// Mitsubishi GX Works2 project: 02fb   PLC: Q03UDV

// task Task_01 (event TRUE, interval 0, priority 31): POU_01
// task st_teste (event TRUE, interval 0, priority 31): st_teste

PROGRAM POU_01
VAR
  CTD_2 : CTD;
  CTU_1 : CTU;
  CTU_2 : CTU;
  R_TRIG_2 : R_TRIG;
  TP_1 : TP;
  TOF_1 : TOF;
  TON_1 : TON;
  timeon : TIME;
  timeof : TIME;
  timetp : TIME;
  TOF_2 : TOF;
  timeof2 : TIME;
  TON_2 : TON;
  timeon2 : TIME;
  TOF_3 : TOF;
  timeof3 : TIME;
  TP_2 : TP;
  TP_3 : TP;
  timept2 : TIME;
  timetp3 : TIME;
  bitOn : BOOL;
  bitOf : BOOL;
  TON_3 : TON;
  TON_4 : TON;
  TON_8 : TON;
  TON5 : TON;
  TOn10 : TON;
  TON_5 : TON;
  timeon5 : TIME;
  timeon3 : TIME;
  TON_6 : TON;
  timeon6 : TIME;
  TOF_4 : TOF;
  timeof7 : TIME;
  verde : BOOL;
  amarelo : BOOL;
  vermelho : BOOL;
  fbBlinker_1 : fbBlinker;
  fbBlinker_2 : fbBlinker;
  diResult : DINT;
  fbBlinker_3 : fbBlinker;
  result : INT;
  funOperacoes_1 : funOperacoes;
  resultS : ARRAY [0..1] OF INT;
  rseultSu : ARRAY [0..1] OF INT;
  resultM : ARRAY [0..1] OF INT;
  resultD : INT;
  resultSo : INT;
  rseultSub : ARRAY [0..1] OF INT;
  resultMult : ARRAY [0..1] OF INT;
  resultMulti : ARRAY [0..1] OF INT;
  resultMultiplicacao : ARRAY [0..1] OF INT;
  resultMUT : ARRAY [0..1] OF INT;
  rseultaSub : ARRAY [0..1] OF INT;
  resultadoSub : ARRAY [0..1] OF INT;
  resultadoMULt : ARRAY [0..1] OF INT;
  Subres : ARRAY [0..1] OF INT;
  Sres : INT;
  Splica : DINT;
  DIVIVALOR : INT;
  Dre : ARRAY [0..1] OF INT;
  habilitar : BOOL;
  valor1 : INT;
  valor2 : INT;
  tipOper : STRING[32];
END_VAR
(* structured ladder/FBD written out as ST: instructions are called as NAME(EN, inputs, outputs); _pN, _eN, _tN stand for wires *)
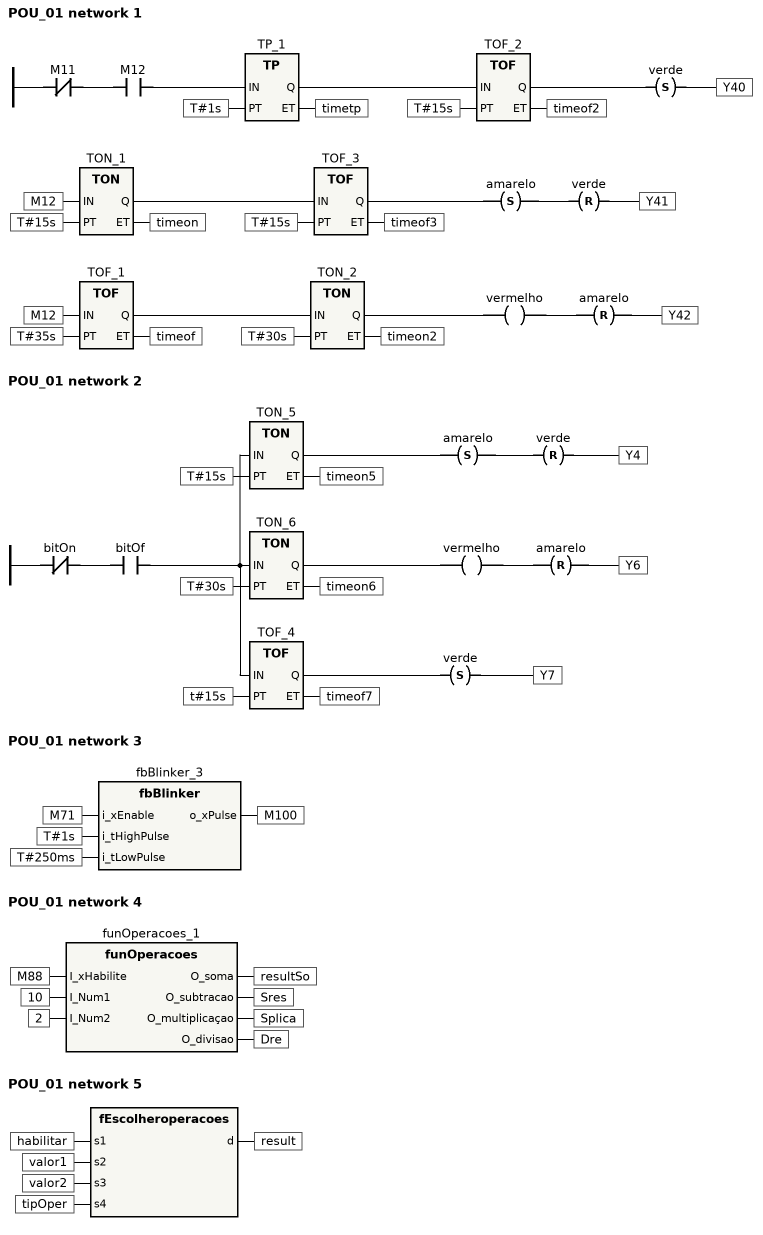
(* network 1 *)
TP_1(IN := NOT M11 AND M12, PT := T#1s, ET => timetp);
TOF_2(IN := TP_1.Q, PT := T#15s, ET => timeof2);
SET(TOF_2.Q, verde);
Y40 := TOF_2.Q;
TON_1(IN := M12, PT := T#15s, ET => timeon);
TOF_3(IN := TON_1.Q, PT := T#15s, ET => timeof3);
SET(TOF_3.Q, amarelo);
RST(TOF_3.Q, verde);
Y41 := TOF_3.Q;
TOF_1(IN := M12, PT := T#35s, ET => timeof);
TON_2(IN := TOF_1.Q, PT := T#30s, ET => timeon2);
vermelho := TON_2.Q;
RST(TON_2.Q, amarelo);
Y42 := TON_2.Q;
(* network 2 *)
_p1 := NOT bitOn AND bitOf;
TOF_4(IN := _p1, PT := t#15s, ET => timeof7);
SET(TOF_4.Q, verde);
Y7 := TOF_4.Q;
TON_5(IN := _p1, PT := T#15s, ET => timeon5);
SET(TON_5.Q, amarelo);
RST(TON_5.Q, verde);
Y4 := TON_5.Q;
TON_6(IN := _p1, PT := T#30s, ET => timeon6);
vermelho := TON_6.Q;
RST(TON_6.Q, amarelo);
Y6 := TON_6.Q;
(* network 3 *)
fbBlinker_3(i_xEnable := M71, i_tHighPulse := T#1s, i_tLowPulse := T#250ms, o_xPulse => M100);
(* network 4 *)
funOperacoes_1(I_xHabilite := M88, I_Num1 := 10, I_Num2 := 2, O_soma => resultSo, O_subtracao => Sres, O_multiplicaçao => Splica, O_divisao => Dre);
(* network 5 *)
result := fEscolheroperacoes(habilitar, valor1, valor2, tipOper);
END_PROGRAM

FUNCTION fSomaInt
VAR_INPUT
  I_xHabilitar : BOOL;
  I_Elemento1 : INT;
  I_Elemento2 : INT;
END_VAR
(* structured ladder/FBD written out as ST: instructions are called as NAME(EN, inputs, outputs); _pN, _eN, _tN stand for wires *)
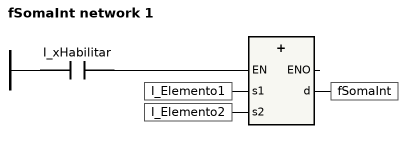
(* network 1 *)
+(I_xHabilitar, I_Elemento1, I_Elemento2, fSomaInt);
END_FUNCTION

FUNCTION fSubtracaoInt
VAR_INPUT
  I_xHabilitarS : BOOL;
  I_Elemento1S : INT;
  I_Elemento2S : INT;
END_VAR
(* structured ladder/FBD written out as ST: instructions are called as NAME(EN, inputs, outputs); _pN, _eN, _tN stand for wires *)
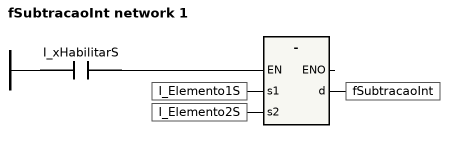
(* network 1 *)
-(I_xHabilitarS, I_Elemento1S, I_Elemento2S, fSubtracaoInt);
END_FUNCTION

FUNCTION_BLOCK fbBlinker
VAR_INPUT
  i_xEnable : BOOL;
  i_tHighPulse : TIME;
  i_tLowPulse : TIME;
END_VAR
VAR_OUTPUT
  o_xPulse : BOOL;
END_VAR
VAR
  fb_TimerHigh : TP;
  fb_TimerLow : TOF;
  xAuxiliar : BOOL;
END_VAR
(* structured ladder/FBD written out as ST: instructions are called as NAME(EN, inputs, outputs); _pN, _eN, _tN stand for wires *)
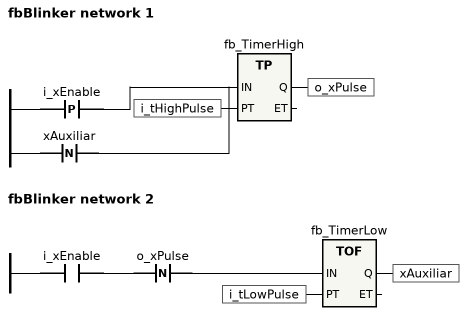
(* network 1 *)
fb_TimerHigh(IN := LDP(TRUE, i_xEnable) OR LDF(TRUE, xAuxiliar), PT := i_tHighPulse, Q => o_xPulse);
(* network 2 *)
fb_TimerLow(IN := i_xEnable AND LDF(TRUE, o_xPulse), PT := i_tLowPulse, Q => xAuxiliar);
END_FUNCTION_BLOCK

FUNCTION fMultInt
VAR_INPUT
  I_xHabilitar : BOOL;
  I_Elemento1 : INT;
  I_Elemento2 : INT;
END_VAR
(* structured ladder/FBD written out as ST: instructions are called as NAME(EN, inputs, outputs); _pN, _eN, _tN stand for wires *)
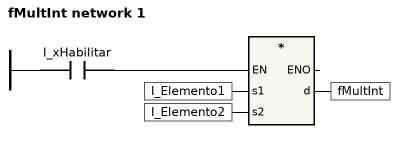
(* network 1 *)
*(I_xHabilitar, I_Elemento1, I_Elemento2, fMultInt);
END_FUNCTION

FUNCTION fDivisaoInt
VAR_INPUT
  I_xHabilitar : BOOL;
  I_Elemento1 : INT;
  I_Elemento2 : INT;
END_VAR
(* structured ladder/FBD written out as ST: instructions are called as NAME(EN, inputs, outputs); _pN, _eN, _tN stand for wires *)
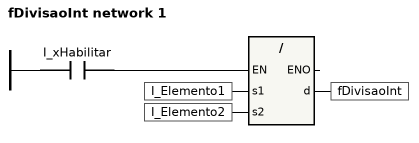
(* network 1 *)
/(I_xHabilitar, I_Elemento1, I_Elemento2, fDivisaoInt);
END_FUNCTION

FUNCTION_BLOCK funOperacoes
VAR_INPUT
  I_xHabilite : BOOL;
  I_Num1 : INT;
  I_Num2 : INT;
END_VAR
VAR_OUTPUT
  O_soma : INT;
  O_subtracao : INT;
  O_multiplicaçao : DINT;
  O_divisao : ARRAY [0..1] OF INT;
END_VAR
VAR
  funOperacoes : INT;
  Dresult : ARRAY [0..1] OF DINT;
  DIVIVALOR : ARRAY [0..1] OF INT;
END_VAR
(* structured ladder/FBD written out as ST: instructions are called as NAME(EN, inputs, outputs); _pN, _eN, _tN stand for wires *)
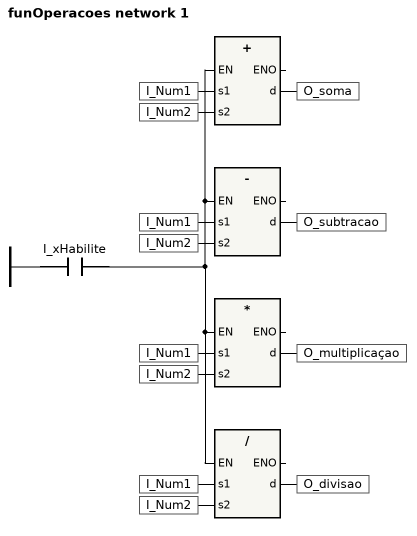
(* network 1 *)
+(I_xHabilite, I_Num1, I_Num2, O_soma);
-(I_xHabilite, I_Num1, I_Num2, O_subtracao);
*(I_xHabilite, I_Num1, I_Num2, O_multiplicaçao);
/(I_xHabilite, I_Num1, I_Num2, O_divisao);
END_FUNCTION_BLOCK

PROGRAM st_teste
VAR
  iRL : ARRAY [0..4] OF INT;
  iRJ : ARRAY [0..4] OF INT;
  iRll : ARRAY [0..9] OF INT;
END_VAR
iRL[1] := fOPcase( TRUE, 5, 2 );
END_PROGRAM

FUNCTION fSoma
VAR_INPUT
  i_Valor1 : INT;
  i_Valor2 : INT;
END_VAR
fSoma:= i_Valor1 + i_Valor2;
END_FUNCTION

FUNCTION fSubt
VAR_INPUT
  i_num1 : INT;
  i_num2 : INT;
END_VAR
fSubt := i_num1 - i_num2;
END_FUNCTION

FUNCTION fMult
VAR_INPUT
  i_n1 : INT;
  i_n2 : INT;
END_VAR
fMult := i_n1* i_n2;
END_FUNCTION

FUNCTION_BLOCK operacoes
VAR_INPUT
  i_1 : INT;
  i_2 : INT;
END_VAR
VAR_OUTPUT
  o_sub : INT;
END_VAR
VAR_INPUT
  o_mult : DINT;
END_VAR
VAR_OUTPUT
  o_soma : INT;
  o_div : ARRAY [0..4] OF INT;
END_VAR
VAR
  operacoes : ARRAY [0..4] OF INT;
  iRs : ARRAY [0..4] OF INT;
END_VAR
operacoes := i_1 , i_2 = fSoma := , fSubt :=  , fMult := , fDiv := ;
END_FUNCTION_BLOCK

FUNCTION fEscolheroperacoes
VAR_INPUT
  xhabilitar : BOOL;
  valor1 : INT;
  valor2 : INT;
  TipOper : STRING[32];
END_VAR
IF xhabilitar THEN 
	IF TipOper="+" THEN 
		fEscolheroperacoes:= valor1 + valor2;
  ELSIF TipOper="-" THEN 
 	fEscolheroperacoes:= valor1 - valor2;
  ELSIF TipOper="*" THEN 
 	fEscolheroperacoes:= valor1 *valor2;
  ELSIF TipOper="/" THEN
 	fEscolheroperacoes:= valor1 / valor2;
  ELSIF ( TipOper="M") OR (TipOper="m") THEN
 	fEscolheroperacoes:= valor1 MOD valor2; 
  ELSE 
 	fEscolheroperacoes:= 32767;
	END_IF;
	
   ELSE 
          fEscolheroperacoes:= -32768;
END_IF;
END_FUNCTION

FUNCTION fDiv
VAR_INPUT
  nu1 : INT;
  nu2 : INT;
END_VAR
fDiv := nu1 / nu2;
END_FUNCTION

FUNCTION fOPcase
VAR_INPUT
  valor1 : INT;
  valor2 : INT;
  xhabilitar : BOOL;
END_VAR
VAR
  auxiliar : ARRAY [0..9] OF INT;
END_VAR
CASE xhabilitar OF
	
	0 : 
	auxiliar[1] := valor1 + valor2; 
	1 :
	auxiliar[2] := valor1 - valor2;
	2 :
	auxiliar[3] := valor1 * valor2;
	3 :
	auxiliar[4] := valor1 / valor2;
	
	ELSE 
	auxiliar[0] := 199;

IF xhabilitar THEN 
   IF auxiliar[1] := "+" THEN 
        ELSIF auxiliar[2]= valor1 - valor2; 
	auxiliar[2] := "-" THEN 
			ELSIF auxiliar[3]= valor1 * valor2;
	auxiliar[3] := "*" THEN 
			ELSIF auxiliar[4]= valor1 / valor2;
		auxiliar[4]	:= "/" THEN 	
ELSIF 	
	auxiliar := 32767;
END_IF 

ELSIF 
	auxiliar : -32767;
	END_IF 
		
END_CASE
END_FUNCTION
